# EPICS substitutions: db/ecmcDS.substitutions
file ecmcDataStorageNew.template
{
  pattern {Index, NELM, T_SMP_MS }
          {1,     100,  -1       }
}
